{attribute addProperty BoxType "EP6228-0022-0016"}
{attribute addProperty Id "Module_1_DeviceState_Inputs_DeviceModule_1_DeviceState_Inputs_Device_50DD3C951620Module_2_DeviceState_InputsModule_2_DeviceState_Inputs_EC75726C6480WcStateAT %I*WcState_F855686C1620InfoDataAT %I*InfoData_275E3363128160"}
{attribute addProperty CRC "1509647662"}
{attribute addProperty SizeInBites "224"}
{attribute addProperty SizeInBytes "28"}
TYPE EP6228_2A1F57FC :
STRUCT
	{attribute addProperty Name "Module_1_DeviceState_Inputs_Device"}
	Module_1_DeviceState_Inputs_Device : Module_1_DeviceState_Inputs_Device_50DD3C95;
	{attribute addProperty Name "Module_2_DeviceState_Inputs"}
	Module_2_DeviceState_Inputs : Module_2_DeviceState_Inputs_EC75726C;
	{attribute addProperty Name "WcState"}
	WcState : WcState_F855686C;
	{attribute addProperty Name "InfoData"}
	InfoData : InfoData_275E3363;
END_STRUCT
END_TYPE

(* stored: Version 1.2.0.0, ProductVersion 3.1.4024.9
   DUT EP6228_2A1F57FC: Id {ef4e70d4-7dfa-4c93-aa7c-021ca98dd51d} *)
